FUNCTION_BLOCK StopMoverGroup  IMPLEMENTS I_Task
VAR
	groupStop			: MC_GroupStop;
	_caGroup			: I_CollisionGroup;
	_Done 				: BOOL;
	_Error				: BOOL;
	_ErrorID			: UDINT;
END_VAR

{analysis -2}

METHOD Abort : BOOL
groupStop.Execute := FALSE;
Abort := TRUE;
END_METHOD

PROPERTY Busy : BOOL
GET
Busy := groupStop.Busy;
END_GET
END_PROPERTY

METHOD Cycle : HRESULT
VAR_INPUT
END_VAR
IF _caGroup = 0 THEN
	cycle := -1;
	RETURN;
END_IF
_Done := groupStop.Done OR _Done;
_Error := groupStop.Error OR _Error;
IF groupStop.ErrorId <> 0 THEN
	_ErrorId := groupStop.ErrorId;
END_IF
groupStop(AxesGroup := _caGroup.GroupRef);
groupStop.Execute := FALSE;
END_METHOD

PROPERTY PUBLIC Deceleration : MC_LREAL
GET
Deceleration := groupStop.Deceleration;
END_GET
SET
IF Deceleration > 0.0 THEN
	groupStop.Deceleration := Deceleration;
END_IF
END_SET
END_PROPERTY

PROPERTY Done : BOOL
GET
Done := _Done;
END_GET
END_PROPERTY

PROPERTY Error : BOOL
GET
Error := _Error;
END_GET
END_PROPERTY

METHOD Execute : HRESULT
IF groupStop.Execute THEN
	Execute := -1;
	RETURN;
END_IF

IF _caGroup = 0 THEN
	Execute := -2;
	RETURN;
END_IF

groupStop.Execute := TRUE;
END_METHOD

PROPERTY PUBLIC Jerk : MC_LREAL
GET
Jerk := groupStop.Jerk;
END_GET
SET
IF Jerk > 0.0 THEN
	groupStop.Jerk := Jerk;
END_IF
END_SET
END_PROPERTY

PROPERTY MyCollisionGroup : I_CollisionGroup
GET
MyCollisionGroup := _caGroup;
END_GET
SET
IF MyCollisionGroup <> 0 THEN
	_caGroup := MyCollisionGroup;
END_IF
END_SET
END_PROPERTY

END_FUNCTION_BLOCK

(* stored: Version 1.1.0.1
   POU StopMoverGroup: Id {1c1e07aa-be1f-4f5f-9f83-11f52cae0c47}, SpecialFunc None
   Method Abort: Id {c537197c-b147-4abf-b878-34be8d4864fb}
   Property Busy: Id {9ebae655-1de1-4c1a-bbd5-86026ed197c9}
   Get Get: Id {a523b092-8918-4349-80ca-f3d4fd4fbef4}
   Method Cycle: Id {eb283c73-ef4f-42f6-83b9-10b77e01e97b}
   Property Deceleration: Id {4b0f086c-1d53-44e4-86b9-9d4a701184a7}
   Get Get: Id {b0811cfb-bb5c-42b5-9a5c-793a076794d1}
   Set Set: Id {d5d2a280-9e98-49b7-b6fe-a592814414dd}
   Property Done: Id {ea125ffd-4438-4a45-8dad-222a40534e69}
   Get Get: Id {5559718d-4e30-4239-9d2e-7f36403bd16b}
   Property Error: Id {d40ba66c-b9b5-460e-90ab-8f59bded3fe6}
   Get Get: Id {812b6ee7-37ac-4dc9-8513-82b9fdd24c3e}
   Method Execute: Id {699db21e-cd5b-48cd-b391-3ef65bad1290}
   Property Jerk: Id {753822d2-3240-4ac1-a838-285435826cfe}
   Get Get: Id {8ec059f8-9a70-4be4-bfe0-899344b2368e}
   Set Set: Id {1e87f5ff-9029-43fd-96bd-fd5c4e284768}
   Property MyCollisionGroup: Id {cb0f23e2-035b-4579-8b52-c9ccb0257f5c}
   Get Get: Id {38655085-d38f-4fef-8c73-780213a29125}
   Set Set: Id {a086e748-ccfd-4e70-a062-66778ac8e3ed} *)
